FUNCTION_BLOCK FB_ShipSimulator
VAR_INPUT
	timestep : LREAL := 0.001;
	
	// Default wavespectrum(Hs=8.0, T1=12.0, spec='JONSWAP')
    w0 : LREAL :=  0.43567172549;
    lambda : LREAL :=  0.101904641875;
    sigma : LREAL :=  5.3310138243;
	
	// PD Contoroller poles
	poles : LREAL := 0.3;
	
	// Max output states allowed
	surge_max : LREAL := 0.2;
	sway_max : LREAL := 0.2;
	heave_max : LREAL := 0.4;
	roll_max : LREAL := 5.0/180.0*pi;
	pitch_max : LREAL := 5.0/180.0*pi;
	yaw_max : LREAL := 5.0/180.0*pi;
	
	
END_VAR
VAR_OUTPUT
	t : LREAL := 0.0;
	
	surge : LREAL;
	sway : LREAL;
	heave : LREAL;
	roll : LREAL;
	pitch : LREAL;
	yaw : LREAL;
END_VAR
VAR
	// Counter variable
	dof : UINT;
	
	// Random generator, initialized in FB_init
	rand : DRAND;

	//  Ship 1st order dynamics from system identification
	Ts_x : LREAL := 45.215;
    Ts_y : LREAL := 18.335;
    Ts_yaw : LREAL := 16.425;
    K_x : LREAL := 1.49944614059E-07;
    K_y : LREAL := 1.13435297558E-07;
    K_yaw : LREAL := 2.77309521498E-10;
	
	// State vectors
	states : ARRAY [0..23] OF LREAL;
	eta : ARRAY [0..5] OF LREAL;
	
	// Scaling gains
	eta_max : ARRAY [0..5] OF LREAL;
	Ks : ARRAY [0..5] OF LREAL := [1.0, 1.0, 1.0, 1.0, 1.0, 1.0];
END_VAR

// Integrate solution by one timestep
integrate();

// Red max settings
eta_max[0] := ABS(surge_max);
eta_max[1] := ABS(sway_max);
eta_max[2] := ABS(heave_max);
eta_max[3] := ABS(roll_max);
eta_max[4] := ABS(pitch_max);
eta_max[5] := ABS(yaw_max);

// Adapt output to fit defined maximum limits
FOR dof := 0 TO 5 DO
	IF ABS(Ks[dof]*states[dof]) >= ABS(eta_max[dof]) THEN
		IF ABS(states[dof]) <> 0.0 THEN
			Ks[dof] := eta_max[dof]/ABS(states[dof]);
		END_IF	
	END_IF	
END_FOR


surge := Ks[0]*states[0];
sway := Ks[1]*states[1];
heave := Ks[2]*states[2];
roll := Ks[3]*states[3];
pitch := Ks[4]*states[4];
yaw := Ks[5]*states[5];

METHOD FB_init : BOOL
VAR_INPUT
	bInitRetains : BOOL; // if TRUE, the retain variables are initialized (warm start / cold start)
	bInCopyCode : BOOL;  // if TRUE, the instance afterwards gets moved into the copy code (online change)
	
	seed : INT;
END_VAR
// Define seed number for stochastic wave
rand.Seed := seed;
END_METHOD

METHOD PRIVATE integrate : BOOL
VAR_INPUT
END_VAR

VAR
	i : DINT;
	
	states_t : ARRAY [0..23] OF LREAL;
END_VAR


states_t := ode(states);

FOR i := 0 TO 23 DO
	states[i] := states[i] + states_t[i]*timestep;
END_FOR

t := t + timestep;
END_METHOD

METHOD PRIVATE kinematics : ARRAY [0..5] OF LREAL;
VAR_INPUT
	eta : ARRAY [0..5] OF LREAL;
	v : ARRAY [0..5] OF LREAL;
END_VAR

VAR
	eta_t : ARRAY[0..5] OF LREAL;
END_VAR

IF COS(eta[4]) <> 0.0 THEN
	eta_t[0] := -v[1]*(COS(eta[3])*SIN(eta[5])-COS(eta[5])*SIN(eta[3])*SIN(eta[4]))+v[2]*(SIN(eta[3])*SIN(eta[5])+COS(eta[3])*COS(eta[5])*SIN(eta[4]))+v[0]*COS(eta[4])*COS(eta[5]);
	eta_t[1] := v[1]*(COS(eta[3])*COS(eta[5])+SIN(eta[3])*SIN(eta[4])*SIN(eta[5]))-v[2]*(COS(eta[5])*SIN(eta[3])-COS(eta[3])*SIN(eta[4])*SIN(eta[5]))+v[0]*COS(eta[4])*SIN(eta[5]);
	eta_t[2] := -v[0]*SIN(eta[4])+v[2]*COS(eta[3])*COS(eta[4])+v[1]*COS(eta[4])*SIN(eta[3]);
	eta_t[3] := v[3]+(v[5]*COS(eta[3])*SIN(eta[4]))/COS(eta[4])+(v[4]*SIN(eta[3])*SIN(eta[4]))/COS(eta[4]);
	eta_t[4] := v[4]*COS(eta[3])-v[5]*SIN(eta[3]);
	eta_t[5] := (v[5]*COS(eta[3]))/COS(eta[4])+(v[4]*SIN(eta[3]))/COS(eta[4]);
	
	kinematics := eta_t;
END_IF;
END_METHOD

METHOD PRIVATE ode : ARRAY [0..23] OF LREAL
VAR_INPUT
	y : ARRAY [0..23] OF LREAL;
END_VAR

VAR
	// Wave component gains
	K : ARRAY [0..5] OF LREAL := [1E4, 1E4, 4E8, 1E8, 1E5, 1E7];	
	
	// PD Controller gains
	Kp : LREAL;
	Kd : LREAL;	
	
	w : LREAL;
	i : UINT;
	
	eta : ARRAY [0..5] OF LREAL;
	eta_t : ARRAY [0..5] OF LREAL;
	
	v : ARRAY [0..5] OF LREAL;
	v_t : ARRAY [0..5] OF LREAL;
	
	x : ARRAY [0..11] OF LREAL;
	x_t : ARRAY [0..11] OF LREAL;
	
	tau : ARRAY [0..5] OF LREAL;
	tau_wave : ARRAY [0..5] OF LREAL;
	tau_tot : ARRAY [0..5] OF LREAL;

	y_t : ARRAY [0..23] OF LREAL;
END_VAR
// Rigid body states
FOR i := 0 TO 5 DO
	eta[i] := y[i];
	v[i] := y[i+6];
END_FOR; 

// Wave simulation states
FOR i := 0 TO 11 DO
	x[i] := y[i+12];
END_FOR

//*******************************************************************//

// Kinematics
eta_t := kinematics(eta, v);

// Wave forces driven by random process
FOR i := 0 TO 5 DO
	rand();
	w := rand.Num*2.0 - 1.0;
	
	x_t[0 + 2*i] := x[1 + 2*i];
	x_t[1 + 2*i] := 2*w*ABS(lambda*sigma*w0) - w0*w0*x[0 + 2*i] - 2*x[1 + 2*i]*ABS(lambda*w0);
	tau_wave[i] := ABS(K[i])*x[1 + 2*i];	
END_FOR;

// PD Controller for DP simulation in surge, sway and yaw directions
Kp := poles*poles*2.0/K_x;
Kd := (2.0*ABS(poles) - 4.0/Ts_x)/K_x;
tau[0] := -(Kp*eta[0] + Kd*eta_t[0]);

Kp := poles*poles*2.0/K_y;
Kd := (2.0*ABS(poles) - 4.0/Ts_y)/K_y;
tau[1] := -(Kp*eta[1] + Kd*eta_t[1]);

Kp := poles*poles*2.0/K_yaw;
Kd := (2.0*ABS(poles) - 4.0/Ts_yaw)/K_yaw;
tau[5] := -(Kp*eta[5] + Kd*eta_t[5]);


// Total forces
tau_tot[0] := tau[0] + tau_wave[0];
tau_tot[1] := tau[1] + tau_wave[1];
tau_tot[2] := tau[2] + tau_wave[2];
tau_tot[3] := tau[3] + tau_wave[3];
tau_tot[4] := tau[4] + tau_wave[4];
tau_tot[5] := tau[5] + tau_wave[5];

// Rigid ship ODE >> v_t = Minv*(-D*v - G*eta + tau + tau_wave)
v_t[0] := 0.000000146900537469*tau_tot[0] - 1.15779191741*eta[4] - 0.00633181020913*eta[2] - 0.000000000481800095922*tau_tot[2] + 0.000000000184278003677*tau_tot[4] - 0.0866236024535*v[0] - 0.00613744736768*v[2] - 0.274323279079*v[4];
v_t[1] := 0.55557891964*eta[3] + 0.000000132912419336*tau_tot[1] - 0.00000000415239105737*tau_tot[3] + 0.0000000000224611856126*tau_tot[5] - 0.253122582192*v[1] - 0.104731972248*v[3] - 0.980405576225*v[5];
v_t[2] := 0.0000000575501415202*tau_tot[2] - 1.50179843329*eta[4] - 0.000000000481800095922*tau_tot[0] - 0.772453112071*eta[2] - 0.000000000397149205293*tau_tot[4] + 0.000284105563467*v[0] - 0.0741429429368*v[2] - 1.51936619529*v[4];
v_t[3] := 0.00000000289648823017*tau_tot[3] - 0.00000000415239105737*tau_tot[1] - 0.387542449503*eta[3] + 0.000000000048718802883*tau_tot[5] + 0.00236474400079*v[1] - 0.0922339025763*v[3] + 0.117970498295*v[5];
v_t[4] := 0.000000000184278003677*tau_tot[0] - 0.954371208694*eta[4] - 0.00521932937313*eta[2] - 0.000000000397149205293*tau_tot[2] + 0.000000000151900888631*tau_tot[4] - 0.00010866416697*v[0] - 0.00505911552371*v[2] - 0.226125468221*v[4];
v_t[5] := 0.0000000000224611856126*tau_tot[1] - 0.00651844672092*eta[3] + 0.000000000048718802883*tau_tot[3] + 0.000000000280999799559*tau_tot[5] - 0.0017495572239*v[1] + 0.0115949285132*v[3] - 0.249188054934*v[5];



//*******************************************************************//

// Rigid body states
FOR i := 0 TO 5 DO
	y_t[i] := eta_t[i];
	y_t[i+6] := v_t[i];
END_FOR; 

// Wave simulation states
FOR i := 0 TO 11 DO
	y_t[i+12] := x_t[i];
END_FOR

// Return y_t
ode := y_t;
END_METHOD

END_FUNCTION_BLOCK

(* stored: Version 1.1.0.1, ProductVersion 3.1.4020.12
   POU FB_ShipSimulator: Id {85434e00-1347-4491-8ec3-e6b62d823d0a}, SpecialFunc None
   Method FB_init: Id {ddd63b4f-29d3-45b7-99d6-e67689b58916}
   Method integrate: Id {e39bc7d8-e772-4ea7-92c8-70edc9febc13}
   Method kinematics: Id {4049487d-e70f-4fac-bc42-aabe50acbc7f}
   Method ode: Id {ab802e49-7ed0-46de-bc34-d6e3e0339237} *)
